TYPE ST_CraneHMIData :
STRUCT
	eMode				: E_ControlBoxSwitchMode := E_ControlBoxSwitchMode.Off;
	eRunningState 		: E_RunningStates;
	bStart				: BOOL;
	//bStop				: BOOL;
	bAuto				: BOOL;
	bOn					: BOOL;
	//bManual				: BOOL;
	fJoyX				: REAL := 1.6384E+04;
	fJoyY				: REAL := 1.6384e+04;	
	sStatus				: STRING;
END_STRUCT
END_TYPE

(* stored: Version 1.1.0.1, ProductVersion 3.1.4024.12
   DUT ST_CraneHMIData: Id {0025e163-92c6-4f5a-b57b-78ebc19918a2} *)
